Yaskawa INFORM job: SYNCS1.JBI

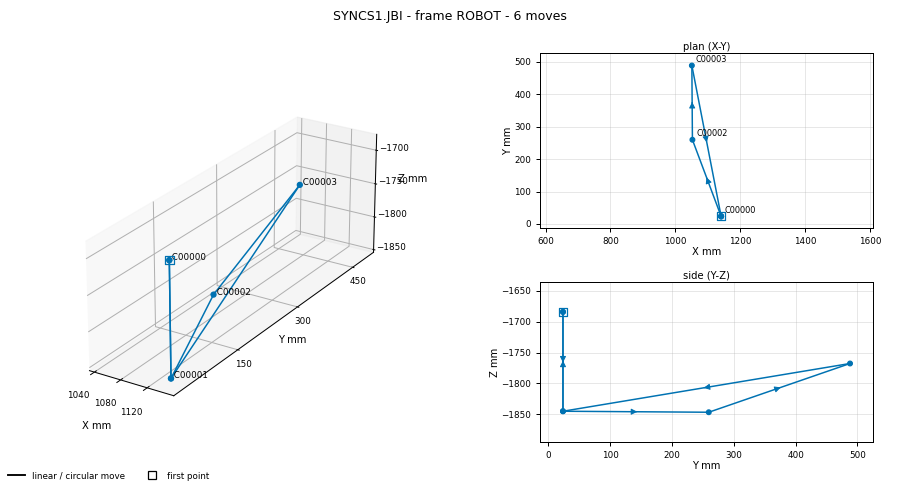
[picture p0: tool path of SYNCS1.JBI in frame ROBOT, 6 of 6 moves have a stored position in this frame; points joined in program order, loops and branches not executed]
/JOB
//NAME SYNCS1
///FOLDERNAME INNE
//POS
///NPOS 6,6,6,0,0,0
///TOOL 0
///POSTYPE ROBOT
///RECTAN
///RCONF 0,0,0,0,0,0,0,0,0,0,0,0,0,0,0,0,0,0,0,0,0,0,0,0
C00000=1141.026,23.497,-1684.152,-5.2688,-0.7428,-80.2434
C00001=1141.027,23.498,-1844.946,-5.2689,-0.7427,-80.2430
C00002=1052.558,259.486,-1846.568,-3.4311,-1.0589,-80.2749
C00003=1050.840,488.131,-1767.664,-4.6109,10.3024,-80.0719
C00004=1141.027,23.498,-1844.946,-5.2689,-0.7427,-80.2430
C00005=1141.026,23.497,-1684.152,-5.2688,-0.7428,-80.2434
BC00000=539.760,812.859,840.896
BC00001=539.760,812.859,840.896
BC00002=539.760,812.859,840.896
BC00003=539.760,812.859,840.896
BC00004=539.760,812.859,840.896
BC00005=539.760,812.859,840.896
///POSTYPE PULSE
///PULSE
EC00000=3,0
EC00001=3,0
EC00002=3,285657
EC00003=118479,285657
EC00004=3,0
EC00005=3,0
//INST
///DATE 2023/10/04 15:16
///ATTR SC,RW,RJ
////FRAME ROBOT
///GROUP1 RB1,BS1
///GROUP2 ST1
NOP
MOVL C00000 BC00000 V=250.0  +MOVJ EC00000 VJ=100.00
PAUSE
MOVL C00001 BC00001 V=75.0  +MOVJ EC00001 VJ=25.00
SMOVL C00002 BC00002 V=75.0  +MOVJ EC00002
SMOVL C00003 BC00003 V=75.0  +MOVJ EC00003
SMOVL C00004 BC00004 V=75.0  +MOVJ EC00004
MOVL C00005 BC00005 V=75.0  +MOVJ EC00005 VJ=25.00
END
